(* IEC 61131-3 sources: Lasal/CPU_5344_V01/Class/Bit2ByteConversion_inputs, 1 file *)

(* ---- Bit2ByteConversion_inputs.st ---- *)
(*!
<Class
	Name               = "Bit2ByteConversion_inputs"
	Revision           = "0.1"
	RealtimeTask       = "false"
	CyclicTask         = "false"
	BackgroundTask     = "false"
	Sigmatek           = "false"
	OSInterface        = "false"
	HighPriority       = "false"
	Automatic          = "false"
	UpdateMode         = "Prescan"
	SharedCommandTable = "true"
	Objectsize         = "(450,2040)">
	<Channels>
		<Server Name="Bit1" Visualized="true" Initialize="false" WriteProtected="false" Retentive="false"/>
		<Server Name="Bit10" Visualized="true" Initialize="false" WriteProtected="false" Retentive="false"/>
		<Server Name="Bit11" Visualized="true" Initialize="false" WriteProtected="false" Retentive="false"/>
		<Server Name="Bit12" Visualized="true" Initialize="false" WriteProtected="false" Retentive="false"/>
		<Server Name="Bit13" Visualized="true" Initialize="false" WriteProtected="false" Retentive="false"/>
		<Server Name="Bit14" Visualized="true" Initialize="false" WriteProtected="false" Retentive="false"/>
		<Server Name="Bit15" Visualized="true" Initialize="false" WriteProtected="false" Retentive="false"/>
		<Server Name="Bit16" Visualized="true" Initialize="false" WriteProtected="false" Retentive="false"/>
		<Server Name="Bit17" Visualized="true" Initialize="false" WriteProtected="false" Retentive="false"/>
		<Server Name="Bit18" Visualized="true" Initialize="false" WriteProtected="false" Retentive="false"/>
		<Server Name="Bit19" Visualized="true" Initialize="false" WriteProtected="false" Retentive="false"/>
		<Server Name="Bit2" Visualized="true" Initialize="false" WriteProtected="false" Retentive="false"/>
		<Server Name="Bit20" Visualized="true" Initialize="false" WriteProtected="false" Retentive="false"/>
		<Server Name="Bit21" Visualized="true" Initialize="false" WriteProtected="false" Retentive="false"/>
		<Server Name="Bit22" Visualized="true" Initialize="false" WriteProtected="false" Retentive="false"/>
		<Server Name="Bit23" Visualized="true" Initialize="false" WriteProtected="false" Retentive="false"/>
		<Server Name="Bit24" Visualized="true" Initialize="false" WriteProtected="false" Retentive="false"/>
		<Server Name="Bit25" Visualized="true" Initialize="false" WriteProtected="false" Retentive="false"/>
		<Server Name="Bit26" Visualized="true" Initialize="false" WriteProtected="false" Retentive="false"/>
		<Server Name="Bit27" Visualized="true" Initialize="false" WriteProtected="false" Retentive="false"/>
		<Server Name="Bit28" Visualized="true" Initialize="false" WriteProtected="false" Retentive="false"/>
		<Server Name="Bit29" Visualized="true" Initialize="false" WriteProtected="false" Retentive="false"/>
		<Server Name="Bit3" Visualized="true" Initialize="false" WriteProtected="false" Retentive="false"/>
		<Server Name="Bit30" Visualized="true" Initialize="false" WriteProtected="false" Retentive="false"/>
		<Server Name="Bit31" Visualized="true" Initialize="false" WriteProtected="false" Retentive="false"/>
		<Server Name="Bit32" Visualized="true" Initialize="false" WriteProtected="false" Retentive="false"/>
		<Server Name="Bit4" Visualized="true" Initialize="false" WriteProtected="false" Retentive="false"/>
		<Server Name="Bit5" Visualized="true" Initialize="false" WriteProtected="false" Retentive="false"/>
		<Server Name="Bit6" Visualized="true" Initialize="false" WriteProtected="false" Retentive="false"/>
		<Server Name="Bit7" Visualized="true" Initialize="false" WriteProtected="false" Retentive="false"/>
		<Server Name="Bit8" Visualized="true" Initialize="false" WriteProtected="false" Retentive="false"/>
		<Server Name="Bit9" Visualized="true" Initialize="false" WriteProtected="false" Retentive="false"/>
		<Server Name="BitValue" Visualized="false" Initialize="false" WriteProtected="false" Retentive="false"/>
		<Client Name="Inv1" Required="false" Internal="false"/>
		<Client Name="Inv10" Required="false" Internal="false"/>
		<Client Name="Inv11" Required="false" Internal="false"/>
		<Client Name="Inv12" Required="false" Internal="false"/>
		<Client Name="Inv13" Required="false" Internal="false"/>
		<Client Name="Inv14" Required="false" Internal="false"/>
		<Client Name="Inv15" Required="false" Internal="false"/>
		<Client Name="Inv16" Required="false" Internal="false"/>
		<Client Name="Inv17" Required="false" Internal="false"/>
		<Client Name="Inv18" Required="false" Internal="false"/>
		<Client Name="Inv19" Required="false" Internal="false"/>
		<Client Name="Inv2" Required="false" Internal="false"/>
		<Client Name="Inv20" Required="false" Internal="false"/>
		<Client Name="Inv21" Required="false" Internal="false"/>
		<Client Name="Inv22" Required="false" Internal="false"/>
		<Client Name="Inv23" Required="false" Internal="false"/>
		<Client Name="Inv24" Required="false" Internal="false"/>
		<Client Name="Inv25" Required="false" Internal="false"/>
		<Client Name="Inv26" Required="false" Internal="false"/>
		<Client Name="Inv27" Required="false" Internal="false"/>
		<Client Name="Inv28" Required="false" Internal="false"/>
		<Client Name="Inv29" Required="false" Internal="false"/>
		<Client Name="Inv3" Required="false" Internal="false"/>
		<Client Name="Inv30" Required="false" Internal="false"/>
		<Client Name="Inv31" Required="false" Internal="false"/>
		<Client Name="Inv32" Required="false" Internal="false"/>
		<Client Name="Inv4" Required="false" Internal="false"/>
		<Client Name="Inv5" Required="false" Internal="false"/>
		<Client Name="Inv6" Required="false" Internal="false"/>
		<Client Name="Inv7" Required="false" Internal="false"/>
		<Client Name="Inv8" Required="false" Internal="false"/>
		<Client Name="Inv9" Required="false" Internal="false"/>
	</Channels>
	<RevDoku>
		<Owner Company="Intecon" Author="Richard Fierkens"/>
		<Dokumentation Revision="0.1" Date="2011-12-28" Author="Richard Fierkens" Company="Intecon" Description="Write timedelay is removed.&#13;&#10;Read timedelay is set to 10mSec."/>
		<Dokumentation Revision="0.0" Date="2011-12-27" Author="Johan Embregts" Company="SigmaControl" Description="Created."/>
	</RevDoku>
</Class>
*)
Bit2ByteConversion_inputs : CLASS
  //Servers:
	BitValue 	: SvrChCmd_BDINT;
	Bit1 	: SvrCh_DINT;
	Bit2 	: SvrCh_DINT;
	Bit3 	: SvrCh_DINT;
	Bit4 	: SvrCh_DINT;
	Bit5 	: SvrCh_DINT;
	Bit6 	: SvrCh_DINT;
	Bit7 	: SvrCh_DINT;
	Bit8 	: SvrCh_DINT;
	Bit9 	: SvrCh_DINT;
	Bit10 	: SvrCh_DINT;
	Bit11 	: SvrCh_DINT;
	Bit12 	: SvrCh_DINT;
	Bit13 	: SvrCh_DINT;
	Bit14 	: SvrCh_DINT;
	Bit15 	: SvrCh_DINT;
	Bit16 	: SvrCh_DINT;
	Bit17 	: SvrCh_DINT;
	Bit18 	: SvrCh_DINT;
	Bit19 	: SvrCh_DINT;
	Bit20 	: SvrCh_DINT;
	Bit21 	: SvrCh_DINT;
	Bit22 	: SvrCh_DINT;
	Bit23 	: SvrCh_DINT;
	Bit24 	: SvrCh_DINT;
	Bit25 	: SvrCh_DINT;
	Bit26 	: SvrCh_DINT;
	Bit27 	: SvrCh_DINT;
	Bit28 	: SvrCh_DINT;
	Bit29 	: SvrCh_DINT;
	Bit30 	: SvrCh_DINT;
	Bit31 	: SvrCh_DINT;
	Bit32 	: SvrCh_DINT;
  //Clients:
	Inv1 	: CltCh_DINT;
	Inv2 	: CltCh_DINT;
	Inv3 	: CltCh_DINT;
	Inv4 	: CltCh_DINT;
	Inv5 	: CltCh_DINT;
	Inv6 	: CltCh_DINT;
	Inv7 	: CltCh_DINT;
	Inv8 	: CltCh_DINT;
	Inv9 	: CltCh_DINT;
	Inv10 	: CltCh_DINT;
	Inv11 	: CltCh_DINT;
	Inv12 	: CltCh_DINT;
	Inv13 	: CltCh_DINT;
	Inv14 	: CltCh_DINT;
	Inv15 	: CltCh_DINT;
	Inv16 	: CltCh_DINT;
	Inv17 	: CltCh_DINT;
	Inv18 	: CltCh_DINT;
	Inv19 	: CltCh_DINT;
	Inv20 	: CltCh_DINT;
	Inv21 	: CltCh_DINT;
	Inv22 	: CltCh_DINT;
	Inv23 	: CltCh_DINT;
	Inv24 	: CltCh_DINT;
	Inv25 	: CltCh_DINT;
	Inv26 	: CltCh_DINT;
	Inv27 	: CltCh_DINT;
	Inv28 	: CltCh_DINT;
	Inv29 	: CltCh_DINT;
	Inv30 	: CltCh_DINT;
	Inv31 	: CltCh_DINT;
	Inv32 	: CltCh_DINT;
  //Variables:
		tMark 	: UDINT;
  //Functions:

	FUNCTION VIRTUAL GLOBAL Init;

	FUNCTION VIRTUAL GLOBAL BitValue::Write
		VAR_INPUT
			input (EAX) 	: BDINT;
		END_VAR
		VAR_OUTPUT
			result (EAX) 	: BDINT;
		END_VAR;
  //Tables:
	FUNCTION @STD
		VAR_OUTPUT
			ret_code	: CONFSTATES;
		END_VAR;
	FUNCTION GLOBAL TAB @CT_;
END_CLASS;

FUNCTION VIRTUAL GLOBAL Bit2ByteConversion_inputs::BitValue::Write
	VAR_INPUT
		input (EAX) 	: BDINT;
	END_VAR
	VAR_OUTPUT
		result (EAX) 	: BDINT;
	END_VAR

	BitValue := input;

  Inv1 := Inv1.Read();
  Inv2 := Inv2.Read();
  Inv3 := Inv3.Read();
  Inv4 := Inv4.Read();
  Inv5 := Inv5.Read();
  Inv6 := Inv6.Read();
  Inv7 := Inv7.Read();
  Inv8 := Inv8.Read();
  Inv9 := Inv9.Read();
  Inv10 := Inv10.Read();
  Inv11 := Inv11.Read();
  Inv12 := Inv12.Read();
  Inv13 := Inv13.Read();
  Inv14 := Inv14.Read();
  Inv15 := Inv15.Read();
  Inv16 := Inv16.Read();
  Inv17 := Inv17.Read();
  Inv18 := Inv18.Read();
  Inv19 := Inv19.Read();
  Inv20 := Inv20.Read();
  Inv21 := Inv21.Read();
  Inv22 := Inv22.Read();
  Inv23 := Inv23.Read();
  Inv24 := Inv24.Read();
  Inv25 := Inv25.Read();
  Inv26 := Inv26.Read();
  Inv27 := Inv27.Read();
  Inv28 := Inv28.Read();
  Inv29 := Inv29.Read();
  Inv30 := Inv30.Read();
  Inv31 := Inv31.Read();
  Inv32 := Inv32.Read();

  Bit1 := abs(BitValue.1 - Inv1);
  Bit2 := abs(BitValue.2 - Inv2);
  Bit3 := abs(BitValue.3 - Inv3);
  Bit4 := abs(BitValue.4 - Inv4);
  Bit5 := abs(BitValue.5 - Inv5);
  Bit6 := abs(BitValue.6 - Inv6);
  Bit7 := abs(BitValue.7 - Inv7);
  Bit8 := abs(BitValue.8 - Inv8);
  Bit9 := abs(BitValue.9 - Inv9);
  Bit10 := abs(BitValue.10 - Inv10);
  Bit11 := abs(BitValue.11 - Inv11);
  Bit12 := abs(BitValue.12 - Inv12);
  Bit13 := abs(BitValue.13 - Inv13);
  Bit14 := abs(BitValue.14 - Inv14);
  Bit15 := abs(BitValue.15 - Inv15);
  Bit16 := abs(BitValue.16 - Inv16);
  Bit17 := abs(BitValue.17 - Inv17);
  Bit18 := abs(BitValue.18 - Inv18);
  Bit19 := abs(BitValue.19 - Inv19);
  Bit20 := abs(BitValue.20 - Inv20);
  Bit21 := abs(BitValue.21 - Inv21);
  Bit22 := abs(BitValue.22 - Inv22);
  Bit23 := abs(BitValue.23 - Inv23);
  Bit24 := abs(BitValue.24 - Inv24);
  Bit25 := abs(BitValue.25 - Inv25);
  Bit26 := abs(BitValue.26 - Inv26);
  Bit27 := abs(BitValue.27 - Inv27);
  Bit28 := abs(BitValue.28 - Inv28);
  Bit29 := abs(BitValue.29 - Inv29);
  Bit30 := abs(BitValue.30 - Inv30);
  Bit31 := abs(BitValue.31 - Inv31);
  Bit32 := abs(BitValue.32 - Inv32);

	result := BitValue;

END_FUNCTION

FUNCTION VIRTUAL GLOBAL Bit2ByteConversion_inputs::Init

  BitValue.Write(input:=0);

END_FUNCTION
